ABB RobotStudio station: Celda - copia.rspag

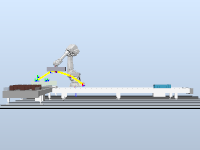
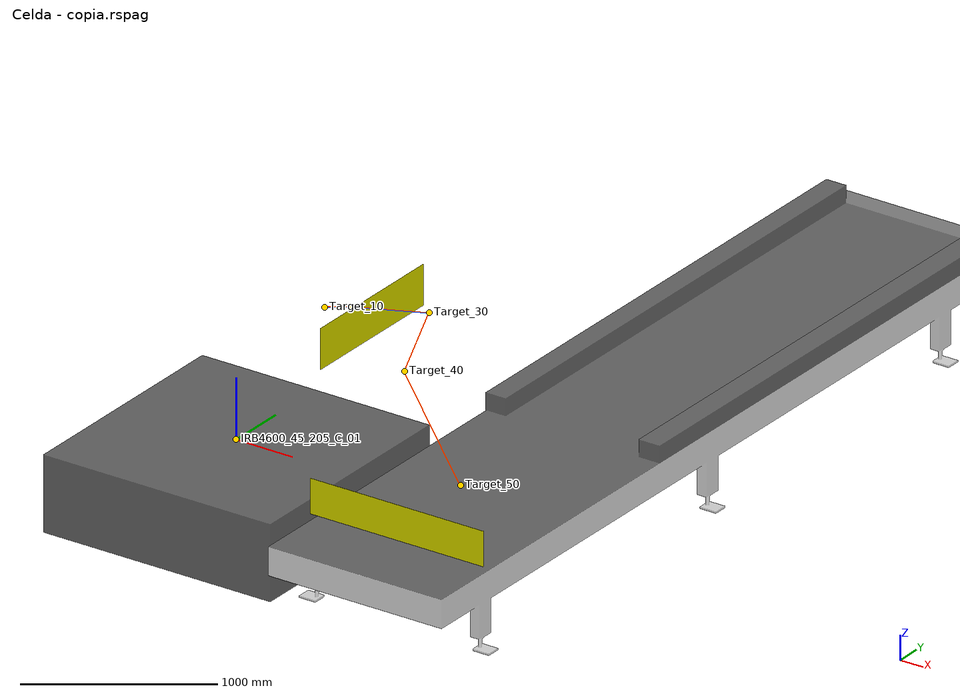
[picture v1: parts stored in the station drawn from their meshes, with robot base, taught points and paths (robot models come from the ABB library and are not in the file)]
--- station ---
Station Celda (saved by RobotStudio 21.3.9648.0)
Controller Controlador1, task T_ROB1: task frame (RAPID world) sits at (0, 0, 435) mm in the station
Controller Controlador1
  mechanical unit ROB_1: IRB4600_45_205_C_01, 6 joints, base frame (0, 0, 0) mm
Layout (positions relative to the parent item):
  - Entrada de canastillas [smart component]
      signals: DO Canasta_ok, DI Soltar, DI Agarrar, DO Agarrado
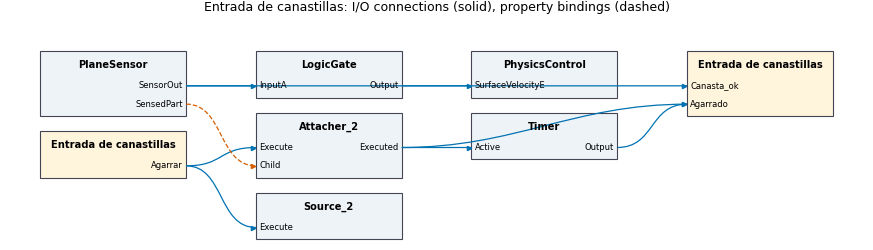
      connections:
        PlaneSensor.SensorOut -> LogicGate.InputA
        LogicGate.Output -> PhysicsControl.SurfaceVelocityEnabled
        PlaneSensor.SensorOut -> Entrada de canastillas.Canasta_ok
        Entrada de canastillas.Agarrar -> Attacher_2.Execute
        Entrada de canastillas.Agarrar -> Source_2.Execute
        Attacher_2.Executed -> Timer.Active
        Timer.Output -> Entrada de canastillas.Agarrado
        Attacher_2.Executed -> Entrada de canastillas.Agarrado
        PlaneSensor.SensedPart => Attacher_2.Child
    - Source_2 [smart component, from Components\Source.rslib]
        properties: Source=Plastic crate; Copy=(none); Parent=(none); Position=[-3.8 1.3 0.565]; Orientation=[3.14159265358979 0 0]; Transient=false; PhysicsBehavior=3
    - PlaneSensor [smart component, from Components\PlaneSensor.rslib]
        properties: Origin=[-0.076705 1.76 0.467165]; Axis1=[0 -0.91 0]; Axis2=[-5E-06 0 0.232835]; SensedPart=(none)
      - _sensorPart_ [part], size 0 x 910 x 232.8 mm
    - PhysicsControl [smart component, from Components\PhysicsControl.rslib]
        properties: Object=Banda_Canastas; Behavior=2; SurfaceVelocity=0.5
    - LogicGate [smart component, from Components\LogicGate.rslib]
        properties: Operator=NOT; Delay=0
    - Attacher_2 [smart component, from Components\Attacher.rslib]
        properties: Parent=MyNewTool; Flange=0; Child=(none); Mount=false; Offset=[0 0 0]; Orientation=[0 0 0]
  - IRB4600_45_205_C_01 [mechanism, from Robots\IRB4600_45_205_C_G_01.rslib] at (0, 0, 435) mm; joint values [0.7854, -0.0486, 0.7239, 0, 0.8955, -2.3562] (rad or m)
  - MyNewTool [mechanism] at (700, 700, 1230.44) mm, rotated rx -180 ry 0 rz 0 deg
      TCP Gripper at (0, 0, 166) mm
      links: NewGripper
  - Perimetro [graphiccomponentgroup]
    - Fence_2503 [graphiccomponentgroup, from Equipment\Fence_2500.rslib] at (3000, 238.8, 0) mm
      - Body 1 [part, from Equipment\Fence_2500.rslib]
      - Body 2 [part, from Equipment\Fence_2500.rslib]
    - Fence_2502 [graphiccomponentgroup, from Equipment\Fence_2500.rslib] at (3000, -2235.69, 0) mm
      - Body 1 [part, from Equipment\Fence_2500.rslib]
      - Body 2 [part, from Equipment\Fence_2500.rslib]
    - Fence_2500 [graphiccomponentgroup, from Equipment\Fence_2500.rslib] at (-2079.28, 2740, 0) mm, rotated rx 0 ry 0 rz -90 deg
      - Body 1 [part, from Equipment\Fence_2500.rslib]
      - Body 2 [part, from Equipment\Fence_2500.rslib]
    - Fence_740_12 [graphiccomponentgroup, from Equipment\Fence_740.rslib] at (3000, -2297.98, 0) mm, rotated rx 0 ry 0 rz 90 deg
      - Body 1 [part, from Equipment\Fence_740.rslib]
      - Body 2 [part, from Equipment\Fence_740.rslib]
    - Fence_740_11 [graphiccomponentgroup, from Equipment\Fence_740.rslib] at (-2100, -2267.47, 0) mm
      - Body 1 [part, from Equipment\Fence_740.rslib]
      - Body 2 [part, from Equipment\Fence_740.rslib]
    - Fence_740_10 [graphiccomponentgroup, from Equipment\Fence_740.rslib] at (82.68, -2200, 0) mm, rotated rx 0 ry 0 rz -90 deg
      - Body 1 [part, from Equipment\Fence_740.rslib]
      - Body 2 [part, from Equipment\Fence_740.rslib]
    - Fence_740_9 [graphiccomponentgroup, from Equipment\Fence_740.rslib] at (-657.15, -2200, 0) mm, rotated rx 0 ry 0 rz -90 deg
      - Body 1 [part, from Equipment\Fence_740.rslib]
      - Body 2 [part, from Equipment\Fence_740.rslib]
    - Fence_740_8 [graphiccomponentgroup, from Equipment\Fence_740.rslib] at (-1386.41, -2200, 0) mm, rotated rx 0 ry 0 rz -90 deg
      - Body 1 [part, from Equipment\Fence_740.rslib]
      - Body 2 [part, from Equipment\Fence_740.rslib]
    - Fence_740_4 [graphiccomponentgroup, from Equipment\Fence_740.rslib] at (-2153.49, -2200, 0) mm, rotated rx 0 ry 0 rz -90 deg
      - Body 1 [part, from Equipment\Fence_740.rslib]
      - Body 2 [part, from Equipment\Fence_740.rslib]
    - Fence_740_3 [graphiccomponentgroup, from Equipment\Fence_740.rslib] at (-2100, -1490.03, 0) mm
      - Body 1 [part, from Equipment\Fence_740.rslib]
      - Body 2 [part, from Equipment\Fence_740.rslib]
    - Fence_740_2 [graphiccomponentgroup, from Equipment\Fence_740.rslib] at (3000, 2740, 0) mm, rotated rx 0 ry 0 rz 90 deg
      - Body 1 [part, from Equipment\Fence_740.rslib]
      - Body 2 [part, from Equipment\Fence_740.rslib]
    - Fence_740 [graphiccomponentgroup, from Equipment\Fence_740.rslib] at (-2100, 2000, 0) mm
      - Body 1 [part, from Equipment\Fence_740.rslib]
      - Body 2 [part, from Equipment\Fence_740.rslib]
    - Gate [graphiccomponentgroup, from Equipment\Fence_Gate.rslib] at (-2100, 728.56, 0) mm, rotated rx 0 ry 0 rz 180 deg
      - Body 1 [part, from Equipment\Fence_Gate.rslib]
      - Body 2 [part, from Equipment\Fence_Gate.rslib]
      - Body 3 [part, from Equipment\Fence_Gate.rslib]
    - Part_2 [part] at (-700, -700, 0) mm, size 1400 x 1400 x 435 mm
  - Plastic crate [part] at (-3299.78, 1300.28, 558.99) mm, rotated rx 179.83 ry 0.16 rz 0.13 deg, size 603.9 x 403.9 x 145.1 mm
  - Entrada de pallets [smart component]
      connections:
        PlaneSensor.SensorOut -> Source.Execute
        PlaneSensor.SensorOut -> LogicGate.InputA
        LogicGate.Output -> PhysicsControl.SurfaceVelocityEnabled
    - Source [smart component, from Components\Source.rslib]
        properties: Source=Euro Pallet; Copy=(none); Parent=(none); Position=[1.75 2.6 0.44]; Orientation=[0 0 1.5707963267949]; Transient=false; PhysicsBehavior=3
    - PlaneSensor [smart component, from Components\PlaneSensor.rslib]
        properties: Origin=[0.84 -0.55 0.475]; Axis1=[1.07 0 0]; Axis2=[0 0 0.2]; SensedPart=(none)
      - _sensorPart_ [part], size 1070 x 0 x 200 mm
    - PhysicsControl [smart component, from Components\PhysicsControl.rslib]
        properties: Object=Banda_P_Entrada_S; Behavior=1; SurfaceVelocity=0.5
    - LogicGate [smart component, from Components\LogicGate.rslib]
        properties: Operator=NOT; Delay=0
  - Bandas [graphiccomponentgroup]
    - Banda_Canastas [part, from Equipment\Conveyor 950 4800 h2.rslib] at (-4200, 850, 0) mm
    - Banda_P_Entrada [part] at (900, 4000, 0) mm, rotated rx 0 ry 0 rz -90 deg, size 5049.9 x 1178.5 x 441.9 mm
    - Banda_P_Entrada_S [part], size 1070 x 4920 x 1 mm
    - Banda_P_Salida [part, from Equipment\Conveyor 950 4000 h2.rslib] at (900, -1050, 0) mm, rotated rx 0 ry 0 rz -90 deg
    - Barrera1 [part], size 130 x 3000 x 100 mm
    - Barrera2 [part] at (-2, 0, 0) mm, size 123 x 3000 x 100 mm
  - Euro Pallet [graphiccomponentgroup, from Equipment\Euro Pallet.rslib] at (1770.21, 2700.56, 450.15) mm, rotated rx 0 ry 0.03 rz 90.01 deg
    - Body 1 [part, from Equipment\Euro Pallet.rslib]
Attachment: MyNewTool is attached to IRB4600_45_205_C_01 / Link6
Station signals: DO Canasta_ok
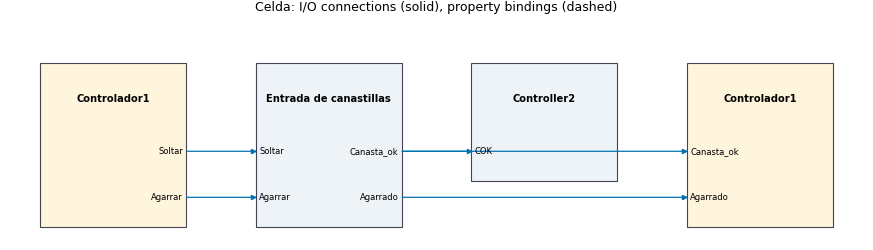
Station logic (signal -> signal, property => property):
  Entrada de canastillas.Canasta_ok -> Controller2.COK
  Entrada de canastillas.Canasta_ok -> Controlador1.Canasta_ok
  Controlador1.Soltar -> Entrada de canastillas.Soltar
  Controlador1.Agarrar -> Entrada de canastillas.Agarrar
  Entrada de canastillas.Agarrado -> Controlador1.Agarrado
Targets, tools, work objects and paths stored in the station and not in the controller backup, written as RAPID:
! task T_ROB1
MODULE Module1
  CONST robtarget Target_60:=[[1570,-267,428],[0,0.707106781,0.707106781,0],[0,0,0,0],[9E+09,9E+09,9E+09,9E+09,9E+09,9E+09]];
  CONST robtarget Target_50_3:=[[1170,333,288],[0,0.707106781,0.707106781,0],[0,0,0,0],[9E+09,9E+09,9E+09,9E+09,9E+09,9E+09]];
  CONST robtarget Target_50_4:=[[1170,-267,288],[0,0.707106781,0.707106781,0],[0,0,0,0],[9E+09,9E+09,9E+09,9E+09,9E+09,9E+09]];
  CONST robtarget Target_50_2:=[[1570,333,288],[0,0.707106781,0.707106781,0],[0,0,0,0],[9E+09,9E+09,9E+09,9E+09,9E+09,9E+09]];
ENDMODULE


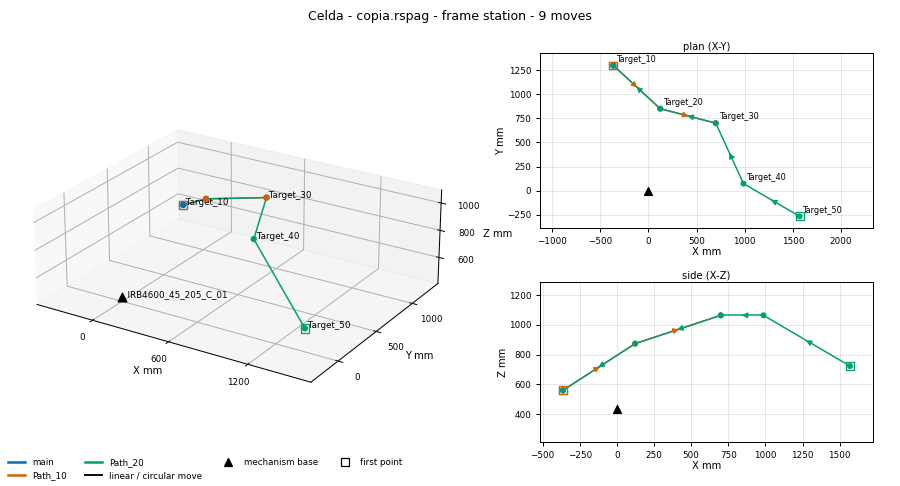
[picture p0: tool path of Celda - copia.rspag in frame station, 9 of 9 moves have a stored position in this frame; points joined in program order, loops and branches not executed]
--- Backups/Controlador1/RAPID/TASK1/PROGMOD/CalibData.mod ---
MODULE CalibData
    PERS tooldata Gripper:=[TRUE,[[0,0,166],[1,0,0,0]],[27.5,[0,0,86.1],[1,0,0,0],0.589498,1.412,1.775]];
    TASK PERS wobjdata Workobject_1:=[FALSE,TRUE,"",[[0,0,0],[1,0,0,0]],[[0,0,0],[1,0,0,0]]];
ENDMODULE

--- Backups/Controlador1/RAPID/TASK1/PROGMOD/Module1.mod ---
MODULE Module1
        CONST robtarget Target_10:=[[-362.824,1298.255,124.558],[0,1,0,0],[0,0,0,0],[9E+09,9E+09,9E+09,9E+09,9E+09,9E+09]];
    CONST robtarget Target_20:=[[123.294942114,850.000075451,439.015995707],[0.000000012,1,-0.000000212,0.000000031],[0,-1,-2,0],[9E+09,9E+09,9E+09,9E+09,9E+09,9E+09]];
    CONST robtarget Target_30:=[[699.999971128,699.99999496,629.43677315],[0.000000004,1,-0.000000218,0.000000007],[0,-1,-2,0],[9E+09,9E+09,9E+09,9E+09,9E+09,9E+09]];
    CONST robtarget Target_50:=[[1570,-267,288],[0,0.707106781,0.707106781,0],[-1,0,0,0],[9E+09,9E+09,9E+09,9E+09,9E+09,9E+09]];
    CONST robtarget Target_40:=[[987.25591454,72.978893792,629.436793547],[0.000000004,-0.699570072,0.714564003,-0.000000013],[0,-1,-1,0],[9E+09,9E+09,9E+09,9E+09,9E+09,9E+09]];
!***********************************************************
    !
    ! Módulo:  Module1
    !
    ! Descripción:
    !   <Introduzca la descripción aquí>
    !
    ! Autor: deste
    !
    ! Versión: 1.0
    !
    !***********************************************************


    !***********************************************************
    !
    ! Procedimiento Main
    !
    !   Este es el punto de entrada de su programa
    !
    !***********************************************************
    PROC main()
        WaitDI Canasta_ok,1;
        MoveL Target_10,v500,z100,Gripper\WObj:=Workobject_1;
        Set Agarrar;
        WaitDI Agarrado,1;
        Path_10;



    ENDPROC
    PROC Path_10()
        MoveL Target_10,v1000,z100,Gripper\WObj:=Workobject_1;
        MoveL Target_20,v1000,z100,Gripper\WObj:=Workobject_1;
        MoveL Target_30,v1000,z100,Gripper\WObj:=Workobject_1;
    ENDPROC
    PROC Path_20()
        MoveL Target_50,v1000,z100,Gripper\WObj:=Workobject_1;
        MoveL Target_40,v1000,z100,Gripper\WObj:=Workobject_1;
        MoveL Target_30,v1000,z100,Gripper\WObj:=Workobject_1;
        MoveL Target_20,v1000,z100,Gripper\WObj:=Workobject_1;
        MoveL Target_10,v1000,z100,Gripper\WObj:=Workobject_1;
    ENDPROC
ENDMODULE

--- Backups/Controlador1/SYSPAR/EIO.cfg ---
EIO:CFG_1.0:6:1::
#
EIO_SIGNAL:

      -Name "Canasta_ok" -SignalType "DI" -Access "All"

      -Name "pallet_ok" -SignalType "DI" -Access "All"

      -Name "Agarrar" -SignalType "DO" -Access "All"

      -Name "Soltar" -SignalType "DO" -Access "All"

      -Name "Agarrado" -SignalType "DI" -Access "All"
